VAR_GLOBAL CONSTANT
	cuintMaxIndex: UINT := 10;
END_VAR

(* stored: Version 1.1.0.1, ProductVersion 3.1.0.23
   GVL Const_CHD: Id {f8ac8dd9-4cd2-46e6-a0c7-1a1ddcabc674} *)
